# EPICS StreamDevice protocol: medipix-ioc/db/devmedipix.proto
##################################################################################
## SOL Group - Diego Dorta - 14/05/2015
##################################################################################
#---------------------------------------------------------------------------------
#---------------------------------------------------------------------------------
ReplyTimeout = 5000;

sendString  	{ out "\$1%s";	in "ok"; @mismatch { in "error"; } }
sendNumber  	{ out "\$1%d";	in "ok"; @mismatch { in "error"; } }
sendCommand 	{ out "\$11";	in "ok"; @mismatch { in "error"; } }
sendReadCounter	{ out "\$1%d";	in "ok"; @mismatch { in "error"; } }
sendGap		{ out "\$1%d";	in "ok"; @mismatch { in "error"; } }

set1  { out "\$1 1"; in "%*150c"; ExtraInput = Ignore; }
set2  { out "\$1 %f"; in "+OMR+%*d+%*d+%*d+%*d+%*d+%*d+%*d+%*d+%*d+%*d+%*d+%*d+%*d+%*d+%*d+%*d+%*d+%*d+%*d+%(\$2)f+%*d+%*f+%*d+"; ExtraInput = Ignore;  }
set3  { out "\$1 %d"; in "+OMR+%*d+%*d+%*d+%*d+%*d+%*d+%*d+%*d+%*d+%*d+%*d+%*d+%*d+%*d+%*d+%*d+%*d+%*d+%*d+%*f+%(\$2)d+%*f+%*d+"; ExtraInput = Ignore;  }
set4  { out "\$1 %d"; in "+OMR+%*d+%*d+%*d+%*d+%*d+%*d+%*d+%*d+%*d+%*d+%*d+%*d+%*d+%*d+%*d+%*d+%*d+%*d+%*d+%*f+%*d+%(\$2)f+%*d+"; ExtraInput = Ignore;  }
set5  { out "\$1 %d"; in "+OMR+%*d+%*d+%*d+%*d+%*d+%*d+%*d+%*d+%*d+%*d+%*d+%*d+%*d+%*d+%*d+%*d+%*d+%*d+%*d+%*f+%*d+%*f+%(\$2)d+"; ExtraInput = Ignore;  }
set6  { out "\$1 %d"; in "+OMR+%*d+%(\$2)d+%*d+%*d+%*d+%*d+%*d+%*d+%*d+%*d+%*d+%*d+%*d+%*d+%*d+%*d+%*d+%*d+%*f+%*f+%*d+%*f+%*d+"; ExtraInput = Ignore;  }
set7  { out "\$1 %d"; in "+OMR+%*d+%*d+%*d+%*d+%*d+%*d+%*d+%*d+%*d+%*d+%*d+%*d+%*d+%(\$2)d+%*d+%*d+%*d+%*d+%*f+%*f+%*d+%*f+%*d+"; ExtraInput = Ignore;  }
set8  { out "\$1 %d"; in "+OMR+%*d+%*d+%(\$2)d+%*d+%*d+%*d+%*d+%*d+%*d+%*d+%*d+%*d+%*d+%*d+%*d+%*d+%*d+%*d+%*f+%*f+%*d+%*f+%*d+"; ExtraInput = Ignore;  }
set9  { out "\$1 %d"; in "+OMR+%*d+%*d+%*d+%*d+%*d+%*d+%*d+%*d+%*d+%*d+%(\$2)d+%*d+%*d+%*d+%*d+%*d+%*d+%*d+%*f+%*f+%*d+%*f+%*d+"; ExtraInput = Ignore;  }
set10 { out "\$1 %d"; in "+OMR+%*d+%*d+%*d+%*d+%*d+%*d+%*d+%*d+%*d+%*d+%*d+%*d+%(\$2)d+%*d+%*d+%*d+%*d+%*d+%*f+%*f+%*d+%*f+%*d+"; ExtraInput = Ignore;  }
set11 { out "\$1 %d"; in "+OMR+%*d+%*d+%*d+%*d+%*d+%*d+%*d+%*d+%*d+%*d+%*d+%*d+%*d+%*d+%*d+%(\$2)d+%*d+%*d+%*f+%*f+%*d+%*f+%*d+"; ExtraInput = Ignore;  }
set12 { out "\$1 %d"; in "+OMR+%*d+%*d+%*d+%*d+%*d+%*d+%(\$2)d+%*d+%*d+%*d+%*d+%*d+%*d+%*d+%*d+%*d+%*d+%*d+%*f+%*f+%*d+%*f+%*d+"; ExtraInput = Ignore;  }
set13 { out "\$1 %d"; in "+OMR+%*d+%*d+%*d+%*d+%*d+%(\$2)d+%*d+%*d+%*d+%*d+%*d+%*d+%*d+%*d+%*d+%*d+%*d+%*d+%*f+%*f+%*d+%*f+%*d+"; ExtraInput = Ignore;  }
set14 { out "\$1 %d"; in "+OMR+%*d+%*d+%*d+%*d+%*d+%*d+%*d+%*d+%*d+%(\$2)d+%*d+%*d+%*d+%*d+%*d+%*d+%*d+%*d+%*f+%*f+%*d+%*f+%*d+"; ExtraInput = Ignore;  }
set15 { out "\$1 %d"; in "+OMR+%*d+%*d+%*d+%*d+%*d+%*d+%*d+%*d+%(\$2)d+%*d+%*d+%*d+%*d+%*d+%*d+%*d+%*d+%*d+%*f+%*f+%*d+%*f+%*d+"; ExtraInput = Ignore;  }
set16 { out "\$1 %d"; in "+OMR+%*d+%*d+%*d+%*d+%(\$2)d+%*d+%*d+%*d+%*d+%*d+%*d+%*d+%*d+%*d+%*d+%*d+%*d+%*d+%*f+%*f+%*d+%*f+%*d+"; ExtraInput = Ignore;  }
set18 { out "\$1 %d"; in "+OMR+%*d+%*d+%*d+%*d+%*d+%*d+%*d+%(\$2)d+%*d+%*d+%*d+%*d+%*d+%*d+%*d+%*d+%*d+%*d+%*d+%*f+%*d+%*f+%*d+"; ExtraInput = Ignore;  }

set19 { out "\$1 %d"; in "+DAC+%(\$2)d+%*d+%*d+%*d+%*d+%*d+%*d+%*d+%*d+%*d+%*d+%*d+%*d+%*d+%*d+%*d+%*d+%*d+%*d+%*d+%*d+%*d+%*d+%*d+%*d+%*d+%*d+"; ExtraInput = Ignore;  }
set20 { out "\$1 %d"; in "+DAC+%*d+%(\$2)d+%*d+%*d+%*d+%*d+%*d+%*d+%*d+%*d+%*d+%*d+%*d+%*d+%*d+%*d+%*d+%*d+%*d+%*d+%*d+%*d+%*d+%*d+%*d+%*d+%*d+"; ExtraInput = Ignore;  }
set21 { out "\$1 %d"; in "+DAC+%*d+%*d+%(\$2)d+%*d+%*d+%*d+%*d+%*d+%*d+%*d+%*d+%*d+%*d+%*d+%*d+%*d+%*d+%*d+%*d+%*d+%*d+%*d+%*d+%*d+%*d+%*d+%*d+"; ExtraInput = Ignore;  }
set22 { out "\$1 %d"; in "+DAC+%*d+%*d+%*d+%(\$2)d+%*d+%*d+%*d+%*d+%*d+%*d+%*d+%*d+%*d+%*d+%*d+%*d+%*d+%*d+%*d+%*d+%*d+%*d+%*d+%*d+%*d+%*d+%*d+"; ExtraInput = Ignore;  }
set23 { out "\$1 %d"; in "+DAC+%*d+%*d+%*d+%*d+%(\$2)d+%*d+%*d+%*d+%*d+%*d+%*d+%*d+%*d+%*d+%*d+%*d+%*d+%*d+%*d+%*d+%*d+%*d+%*d+%*d+%*d+%*d+%*d+"; ExtraInput = Ignore;  }
set24 { out "\$1 %d"; in "+DAC+%*d+%*d+%*d+%*d+%*d+%(\$2)d+%*d+%*d+%*d+%*d+%*d+%*d+%*d+%*d+%*d+%*d+%*d+%*d+%*d+%*d+%*d+%*d+%*d+%*d+%*d+%*d+%*d+"; ExtraInput = Ignore;  }
set25 { out "\$1 %d"; in "+DAC+%*d+%*d+%*d+%*d+%*d+%*d+%(\$2)d+%*d+%*d+%*d+%*d+%*d+%*d+%*d+%*d+%*d+%*d+%*d+%*d+%*d+%*d+%*d+%*d+%*d+%*d+%*d+%*d+"; ExtraInput = Ignore;  }
set26 { out "\$1 %d"; in "+DAC+%*d+%*d+%*d+%*d+%*d+%*d+%*d+%(\$2)d+%*d+%*d+%*d+%*d+%*d+%*d+%*d+%*d+%*d+%*d+%*d+%*d+%*d+%*d+%*d+%*d+%*d+%*d+%*d+"; ExtraInput = Ignore;  }
set27 { out "\$1 %d"; in "+DAC+%*d+%*d+%*d+%*d+%*d+%*d+%*d+%*d+%*d+%(\$2)d+%*d+%*d+%*d+%*d+%*d+%*d+%*d+%*d+%*d+%*d+%*d+%*d+%*d+%*d+%*d+%*d+%*d+"; ExtraInput = Ignore;  }
set28 { out "\$1 %d"; in "+DAC+%*d+%*d+%*d+%*d+%*d+%*d+%*d+%*d+%*d+%*d+%(\$2)d+%*d+%*d+%*d+%*d+%*d+%*d+%*d+%*d+%*d+%*d+%*d+%*d+%*d+%*d+%*d+%*d+"; ExtraInput = Ignore;  }
set29 { out "\$1 %d"; in "+DAC+%*d+%*d+%*d+%*d+%*d+%*d+%*d+%*d+%*d+%*d+%*d+%(\$2)d+%*d+%*d+%*d+%*d+%*d+%*d+%*d+%*d+%*d+%*d+%*d+%*d+%*d+%*d+%*d+"; ExtraInput = Ignore;  }
set30 { out "\$1 %d"; in "+DAC+%*d+%*d+%*d+%*d+%*d+%*d+%*d+%*d+%*d+%*d+%*d+%*d+%(\$2)d+%*d+%*d+%*d+%*d+%*d+%*d+%*d+%*d+%*d+%*d+%*d+%*d+%*d+%*d+"; ExtraInput = Ignore;  }
set31 { out "\$1 %d"; in "+DAC+%*d+%*d+%*d+%*d+%*d+%*d+%*d+%*d+%*d+%*d+%*d+%*d+%*d+%*d+%(\$2)d+%*d+%*d+%*d+%*d+%*d+%*d+%*d+%*d+%*d+%*d+%*d+%*d+"; ExtraInput = Ignore;  }
set32 { out "\$1 %d"; in "+DAC+%*d+%*d+%*d+%*d+%*d+%*d+%*d+%*d+%*d+%*d+%*d+%*d+%*d+%*d+%*d+%*d+%(\$2)d+%*d+%*d+%*d+%*d+%*d+%*d+%*d+%*d+%*d+%*d+"; ExtraInput = Ignore;  }
set33 { out "\$1 %d"; in "+DAC+%*d+%*d+%*d+%*d+%*d+%*d+%*d+%*d+%(\$2)d+%*d+%*d+%*d+%*d+%*d+%*d+%*d+%*d+%*d+%*d+%*d+%*d+%*d+%*d+%*d+%*d+%*d+%*d+"; ExtraInput = Ignore;  }
set34 { out "\$1 %d"; in "+DAC+%*d+%*d+%*d+%*d+%*d+%*d+%*d+%*d+%*d+%*d+%*d+%*d+%*d+%*d+%*d+%*d+%*d+%(\$2)d+%*d+%*d+%*d+%*d+%*d+%*d+%*d+%*d+%*d+"; ExtraInput = Ignore;  }
set35 { out "\$1 %d"; in "+DAC+%*d+%*d+%*d+%*d+%*d+%*d+%*d+%*d+%*d+%*d+%*d+%*d+%*d+%*d+%*d+%*d+%*d+%*d+%(\$2)d+%*d+%*d+%*d+%*d+%*d+%*d+%*d+%*d+"; ExtraInput = Ignore;  }
set36 { out "\$1 %d"; in "+DAC+%*d+%*d+%*d+%*d+%*d+%*d+%*d+%*d+%*d+%*d+%*d+%*d+%*d+%*d+%*d+%*d+%*d+%*d+%*d+%(\$2)d+%*d+%*d+%*d+%*d+%*d+%*d+%*d+"; ExtraInput = Ignore;  }
set37 { out "\$1 %d"; in "+DAC+%*d+%*d+%*d+%*d+%*d+%*d+%*d+%*d+%*d+%*d+%*d+%*d+%*d+%*d+%*d+%*d+%*d+%*d+%*d+%*d+%*d+%(\$2)d+%*d+%*d+%*d+%*d+%*d+"; ExtraInput = Ignore;  }
set38 { out "\$1 %d"; in "+DAC+%*d+%*d+%*d+%*d+%*d+%*d+%*d+%*d+%*d+%*d+%*d+%*d+%*d+%*d+%*d+%*d+%*d+%*d+%*d+%*d+%*d+%*d+%(\$2)d+%*d+%*d+%*d+%*d+"; ExtraInput = Ignore;  }
set39 { out "\$1 %d"; in "+DAC+%*d+%*d+%*d+%*d+%*d+%*d+%*d+%*d+%*d+%*d+%*d+%*d+%*d+%*d+%*d+%*d+%*d+%*d+%*d+%*d+%*d+%*d+%*d+%(\$2)d+%*d+%*d+%*d+"; ExtraInput = Ignore;  }
set40 { out "\$1 %d"; in "+DAC+%*d+%*d+%*d+%*d+%*d+%*d+%*d+%*d+%*d+%*d+%*d+%*d+%*d+%*d+%*d+%*d+%*d+%*d+%*d+%*d+%*d+%*d+%*d+%*d+%(\$2)d+%*d+%*d+"; ExtraInput = Ignore;  }
set41 { out "\$1 %d"; in "+DAC+%*d+%*d+%*d+%*d+%*d+%*d+%*d+%*d+%*d+%*d+%*d+%*d+%*d+%*d+%*d+%*d+%*d+%*d+%*d+%*d+%*d+%*d+%*d+%*d+%*d+%(\$2)d+%*d+"; ExtraInput = Ignore;  }
set42 { out "\$1 %d"; in "+DAC+%*d+%*d+%*d+%*d+%*d+%*d+%*d+%*d+%*d+%*d+%*d+%*d+%*d+%*d+%*d+%*d+%*d+%*d+%*d+%*d+%*d+%*d+%*d+%*d+%*d+%*d+%(\$2)d+"; ExtraInput = Ignore;  }
set43 { out "\$1 %d"; in "+DAC+%*d+%*d+%*d+%*d+%*d+%*d+%*d+%*d+%*d+%*d+%*d+%*d+%*d+%*d+%*d+%*d+%*d+%*d+%*d+%*d+%(\$2)d+%*d+%*d+%*d+%*d+%*d+%*d+"; ExtraInput = Ignore;  }

set44  { out "\$1 %s"; in "%*150c"; @mismatch { in ""; } }
set45  { out "\$1 %d"; in "%*150c"; @mismatch { in ""; } }
set46  { out "\$1 %s"; in "%*150c"; @mismatch { in ""; } }

setRefreshOMR { out "\$1 7";
		in "+OMR+"
			"%*d+"
			"%(\$2:GetCountMode)d+"
			"%(\$2:GetPolarity)d+"
			"%*d+"
			"%(\$2:GetDiscSel)d+"
			"%(\$2:GetEnableTestPulse)d+"
			"%(\$2:GetNumberBitCounter)d+"
			"%(\$2:GetColumNBlock)d+"
			"%(\$2:GetColumBlockSel)d+"
			"%(\$2:GetRowBlock)d+"
			"%(\$2:GetRowBlockSel)d+"
			"%*d+"
			"%(\$2:GetColorMode)d+"
			"%(\$2:GetPixelMode)d+"
			"%*d+"
			"%(\$2:GetGainMode)d+"
			"%*d+"
			"%*d+"
			"%*d+"
			"%(\$3:GetAcquisitionTime)f+"
			"%(\$3:GetNumberFrames)d+"
			"%(\$3:GetGap)f+"
			"%(\$3:GetReadCounter)d+"; ExtraInput = Ignore;  }

setRefreshDAC { out "\$1 6";
		in "+DAC+"
			"%(\$2:GetThreshold_0)d+"
			"%(\$2:GetThreshold_1)d+"
			"%(\$2:GetThreshold_2)d+"
			"%(\$2:GetThreshold_3)d+"
			"%(\$2:GetThreshold_4)d+"
			"%(\$2:GetThreshold_5)d+"
			"%(\$2:GetThreshold_6)d+"
			"%(\$2:GetThreshold_7)d+"
			"%*d+"
			"%*d+"
			"%*d+"
			"%*d+"
			"%*d+"
			"%*d+"
			"%*d+"
			"%*d+"
			"%*d+"
			"%*d+"
			"%*d+"
			"%*d+"
			"%*d+"
			"%*d+"
			"%*d+"
			"%*d+"
			"%*d+"
			"%*d+"
			"%*d+"; ExtraInput = Ignore;  }
